{attribute 'GeneratedUsingTerminal: EL3111-0000-0016'}
{attribute addProperty BoxType "EL3111-0000-0016"}
{attribute addProperty Id "EtcSlaveTerminalBaseAI_StandardAT %I*AI_Standard_A8DF64E310WcStateAT %I*WcState_9091E0EB2InfoDataAT %I*InfoData_32EB74EA10"}
{attribute addProperty CRC "279820378"}
{attribute addProperty Size "22"}
TYPE EL3111_10ADB85A EXTENDS EtcSlaveTerminalBase :
STRUCT
	{attribute addProperty Name "AI_Standard"}
	AI_Standard : AI_Standard_A8DF64E3;
	{attribute addProperty Name "WcState"}
	WcState : WcState_9091E0EB;
	{attribute addProperty Name "InfoData"}
	InfoData : InfoData_32EB74EA;
END_STRUCT
END_TYPE

(* stored: Version 1.2.0.0, ProductVersion 3.1.4024.9
   DUT EL3111_10ADB85A: Id {bcfb030b-ce03-420c-8c99-fca9fd70c30d} *)
